(* Logix 5000 project; controller Drives_Line1 1756-L72 rev 20.13; software revision 20.04; part 17 of 21 *)
(* tags used below, declared in another part *)
   Bridle_04 : UDT_Bridle_3M;
   Bridle_04_FB_Diff : DINT;
   Bridle_04_FB_Update_Valid : BOOL;
   Bridle_04_Rev_mm : REAL;
   Bridle_04b_FBCounts_mm : REAL;
   Exit_Accu : UDT_Exit_Accu;
   ExitCtrl : UDT_Control_Zone;
   In_Config : UDT_Config;
   LineCmd : UDT_Commands_Line;
   Out_Feedbacks : UDT_Fdbks;
   Out_Status : UDT_Status;
   TaskInterval_ms : DINT;
   TestConfig_Exit_Accu : UDT_Config_Accu;
   TM3 : UDT_TM;
   zBridle_04b_Max_rev : REAL;
   zConfigFromMaster : BOOL;
   zPi : REAL;
(* P18_Exit_Accu, continued *)

ROUTINE R98_ToDrive   (* ladder *)
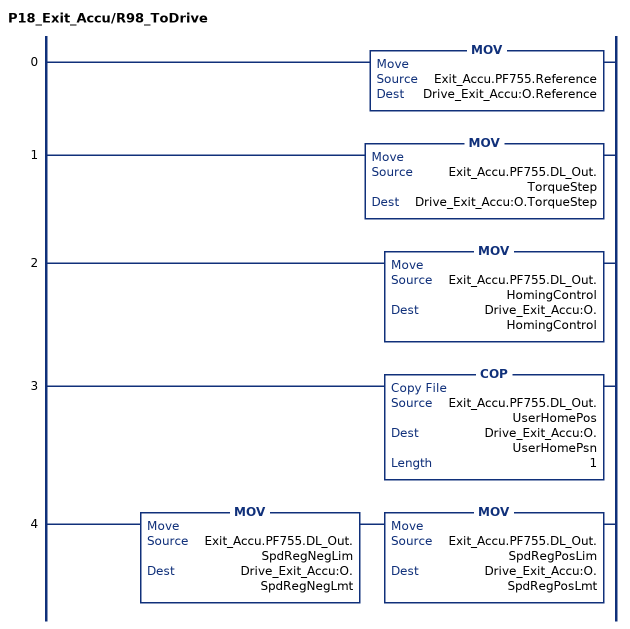
   0: MOV(Exit_Accu.PF755.Reference,Drive_Exit_Accu:O.Reference);
   1: MOV(Exit_Accu.PF755.DL_Out.TorqueStep,Drive_Exit_Accu:O.TorqueStep);
   2: MOV(Exit_Accu.PF755.DL_Out.HomingControl,Drive_Exit_Accu:O.HomingControl);
   3: COP(Exit_Accu.PF755.DL_Out.UserHomePos,Drive_Exit_Accu:O.UserHomePsn,1);
   4: MOV(Exit_Accu.PF755.DL_Out.SpdRegNegLim,Drive_Exit_Accu:O.SpdRegNegLmt)MOV(Exit_Accu.PF755.DL_Out.SpdRegPosLim,Drive_Exit_Accu:O.SpdRegPosLmt);
END_ROUTINE

ROUTINE R999_Test   (* ladder *)
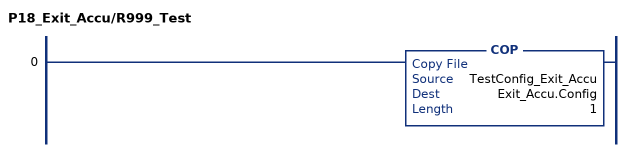
   0: COP(TestConfig_Exit_Accu,Exit_Accu.Config,1);
END_ROUTINE

ROUTINE R99_To_Master   (* ladder *)
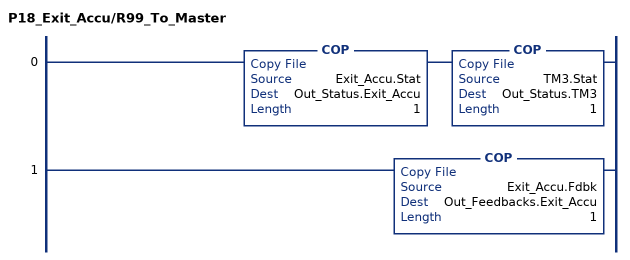
   0: COP(Exit_Accu.Stat,Out_Status.Exit_Accu,1)COP(TM3.Stat,Out_Status.TM3,1);
   1: COP(Exit_Accu.Fdbk,Out_Feedbacks.Exit_Accu,1);
END_ROUTINE
END_PROGRAM

PROGRAM P19_Bridle_04   (* main routine R00_Main *)
VAR
   ADD_01 : FBD_MATH := (SourceA := 0.0679603, Dest := 0.0679603);
   ADD_02 : FBD_MATH;
   BNOT_01 : FBD_BOOLEAN_NOT := (In := 1);
   BNOT_02 : FBD_BOOLEAN_NOT := (Out := 1);
   BOR_01 : FBD_BOOLEAN_OR := (In1 := 1, Out := 1);
   Bridle_04_FB_Count_Old : DINT := 7917204;
   Bridle_04_Max_FBcounts : REAL := 5120.0;
   Bridle_04_SpdTrimMPS : REAL;
   Bridle_04_SpdTrimPct : REAL;
   Bridle_04a_RPMPerMPS : REAL := 3303.7466;
   Bridle_04b_RPMPerMPS : REAL := 3085.579;
   Bridle_04c_RPMPerMPS : REAL := 2662.344;
   DIV_01 : FBD_MATH := (SourceB := 100.0);
   EQU_01 : FBD_COMPARE := (SourceA := 0.084748514);
   IO_State_Bridle_04a : INT := 4;
   IO_State_Bridle_04b : INT := 4;
   IO_State_Bridle_04c : INT := 4;
   IO_State_Tmp_Bridle_04a : INT := 16384;
   IO_State_Tmp_Bridle_04b : INT := 16384;
   IO_State_Tmp_Bridle_04c : INT := 16384;
   MUL_01 : FBD_MATH := (SourceB := 3085.579);
   MUL_02 : FBD_MATH := (SourceB := 3303.7466);
   MUL_05 : FBD_MATH;
   MUL_06 : FBD_MATH := (SourceB := 2662.344);
   Ons : DINT;
   PI_02 : PROP_INT := (In := -2.3841858e-07, Initialize := 1, Kp := 0.25, Wld := 0.05, HighLimit := 2.5, LowLimit := -2.5, ShapeKpPlus := 1.0, ShapeKpMinus := 1.0, ShapeWldPlus := 1.0, ShapeWldMinus := 1.0, RTSTime := 1, DeltaT := 0.05);
   PulsReset_PID : TIMER := (PRE := 250);
   SCL_09 : SCALE := (InRawMax := 100.0, InRawMin := -100.0, InEUMax := 2.5, InEUMin := -2.5, Limiting := 1, Out := -2.3841858e-07);
   SUB_02 : FBD_MATH;
   TimeOn_PIDOn : TIMER := (PRE := 500);
   TofReset : TIMER := (PRE := 1000, ACC := 1000);
   TonNoResponse : TIMER[3] := ([0].PRE := 2500, [1].PRE := 2500, [2].PRE := 2500);
   zBridle_04_Ki_SpdTrim : REAL := 0.05;
   zBridle_04_Kp_SpdTrim : REAL := 0.25;
   zBridle_04_MaxTrimSpdTrim : REAL := 2.5;
   zBridle_04_MinTrimSpdTrim : REAL := -2.5;
   zBridle_04b_EncRes : REAL := 4096.0;
END_VAR

ROUTINE R00_Main   (* ladder *)
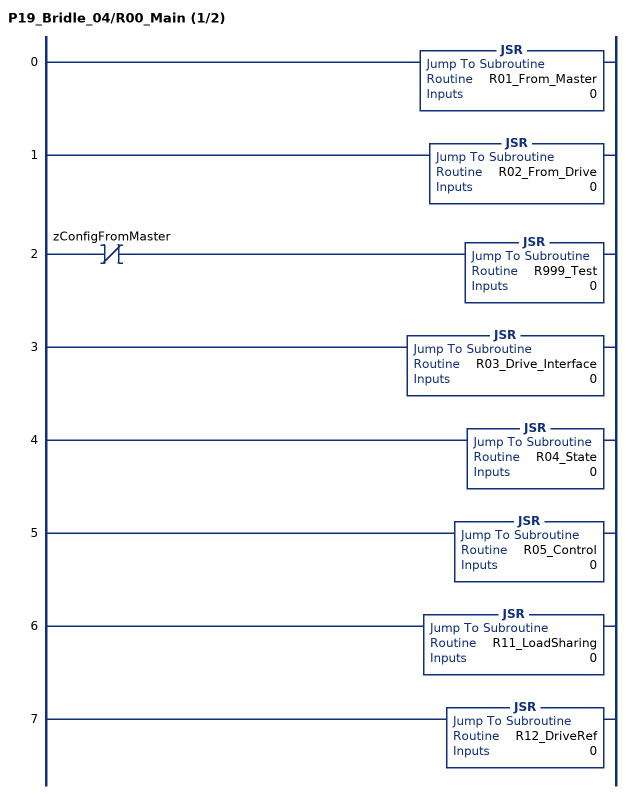
   0: JSR(R01_From_Master,0);
   1: JSR(R02_From_Drive,0);
   2: XIO(zConfigFromMaster)JSR(R999_Test,0);
   3: JSR(R03_Drive_Interface,0);
   4: JSR(R04_State,0);
   5: JSR(R05_Control,0);
   6: JSR(R11_LoadSharing,0);
   7: JSR(R12_DriveRef,0);
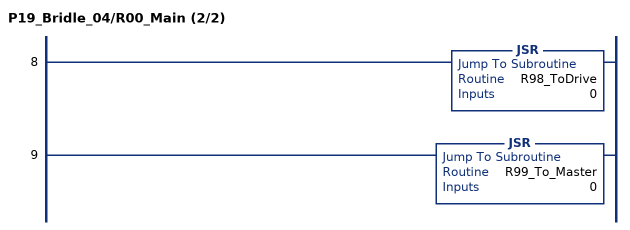
   8: JSR(R98_ToDrive,0);
   9: JSR(R99_To_Master,0);
END_ROUTINE

ROUTINE R01_From_Master   (* ladder *)
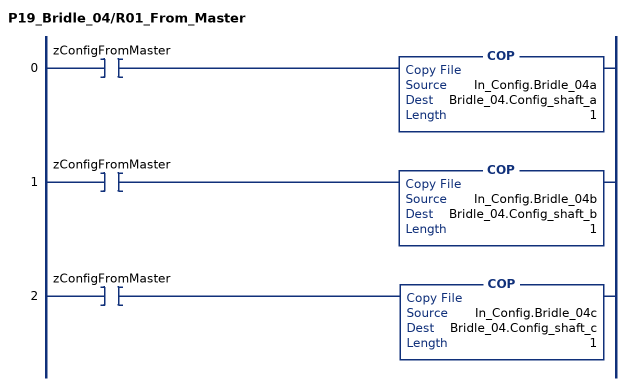
   0: XIC(zConfigFromMaster)COP(In_Config.Bridle_04a,Bridle_04.Config_shaft_a,1);
   1: XIC(zConfigFromMaster)COP(In_Config.Bridle_04b,Bridle_04.Config_shaft_b,1);
   2: XIC(zConfigFromMaster)COP(In_Config.Bridle_04c,Bridle_04.Config_shaft_c,1);
END_ROUTINE

ROUTINE R02_From_Drive   (* ladder *)
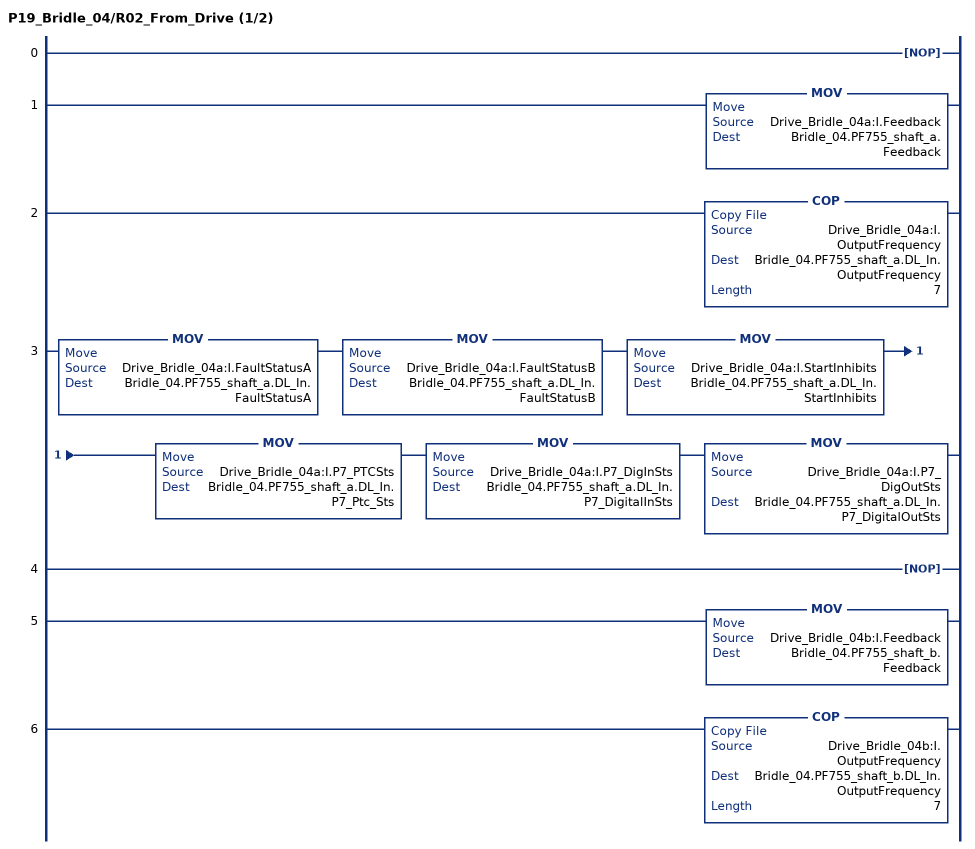
   0: NOP();
   1: MOV(Drive_Bridle_04a:I.Feedback,Bridle_04.PF755_shaft_a.Feedback);
   2: COP(Drive_Bridle_04a:I.OutputFrequency,Bridle_04.PF755_shaft_a.DL_In.OutputFrequency,7);
   3: MOV(Drive_Bridle_04a:I.FaultStatusA,Bridle_04.PF755_shaft_a.DL_In.FaultStatusA)MOV(Drive_Bridle_04a:I.FaultStatusB,Bridle_04.PF755_shaft_a.DL_In.FaultStatusB)MOV(Drive_Bridle_04a:I.StartInhibits,Bridle_04.PF755_shaft_a.DL_In.StartInhibits)MOV(Drive_Bridle_04a:I.P7_PTCSts,Bridle_04.PF755_shaft_a.DL_In.P7_Ptc_Sts)MOV(Drive_Bridle_04a:I.P7_DigInSts,Bridle_04.PF755_shaft_a.DL_In.P7_DigitalInSts)MOV(Drive_Bridle_04a:I.P7_DigOutSts,Bridle_04.PF755_shaft_a.DL_In.P7_DigitalOutSts);
   4: NOP();
   5: MOV(Drive_Bridle_04b:I.Feedback,Bridle_04.PF755_shaft_b.Feedback);
   6: COP(Drive_Bridle_04b:I.OutputFrequency,Bridle_04.PF755_shaft_b.DL_In.OutputFrequency,7);
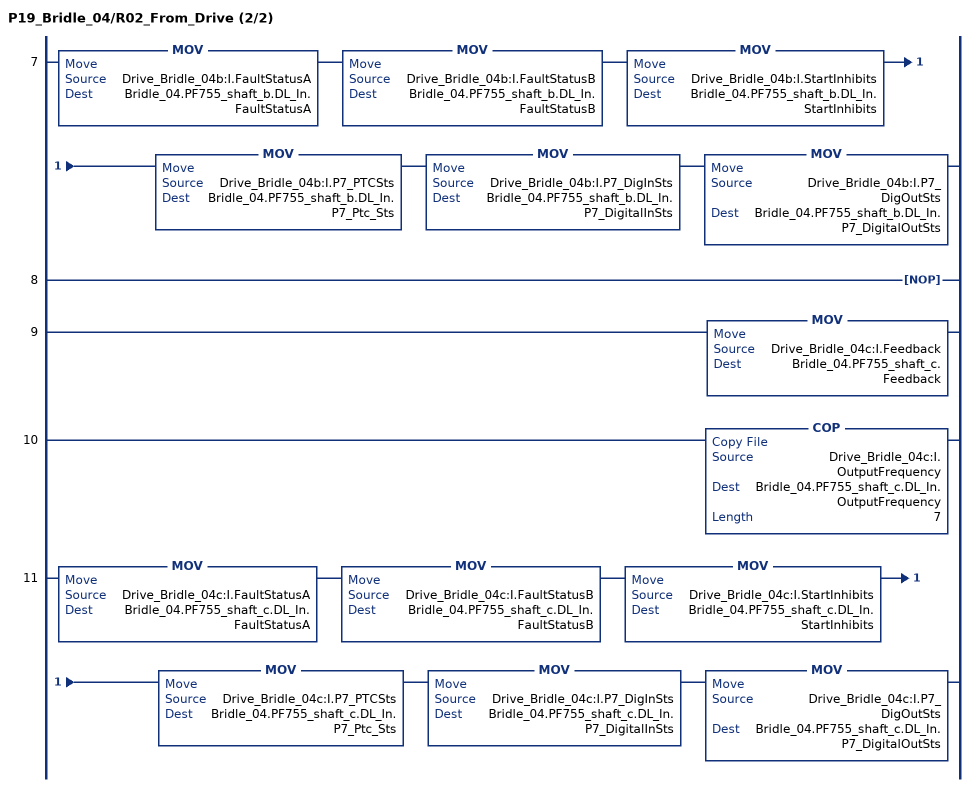
   7: MOV(Drive_Bridle_04b:I.FaultStatusA,Bridle_04.PF755_shaft_b.DL_In.FaultStatusA)MOV(Drive_Bridle_04b:I.FaultStatusB,Bridle_04.PF755_shaft_b.DL_In.FaultStatusB)MOV(Drive_Bridle_04b:I.StartInhibits,Bridle_04.PF755_shaft_b.DL_In.StartInhibits)MOV(Drive_Bridle_04b:I.P7_PTCSts,Bridle_04.PF755_shaft_b.DL_In.P7_Ptc_Sts)MOV(Drive_Bridle_04b:I.P7_DigInSts,Bridle_04.PF755_shaft_b.DL_In.P7_DigitalInSts)MOV(Drive_Bridle_04b:I.P7_DigOutSts,Bridle_04.PF755_shaft_b.DL_In.P7_DigitalOutSts);
   8: NOP();
   9: MOV(Drive_Bridle_04c:I.Feedback,Bridle_04.PF755_shaft_c.Feedback);
   10: COP(Drive_Bridle_04c:I.OutputFrequency,Bridle_04.PF755_shaft_c.DL_In.OutputFrequency,7);
   11: MOV(Drive_Bridle_04c:I.FaultStatusA,Bridle_04.PF755_shaft_c.DL_In.FaultStatusA)MOV(Drive_Bridle_04c:I.FaultStatusB,Bridle_04.PF755_shaft_c.DL_In.FaultStatusB)MOV(Drive_Bridle_04c:I.StartInhibits,Bridle_04.PF755_shaft_c.DL_In.StartInhibits)MOV(Drive_Bridle_04c:I.P7_PTCSts,Bridle_04.PF755_shaft_c.DL_In.P7_Ptc_Sts)MOV(Drive_Bridle_04c:I.P7_DigInSts,Bridle_04.PF755_shaft_c.DL_In.P7_DigitalInSts)MOV(Drive_Bridle_04c:I.P7_DigOutSts,Bridle_04.PF755_shaft_c.DL_In.P7_DigitalOutSts);
END_ROUTINE

ROUTINE R03_Drive_Interface   (* ladder *)
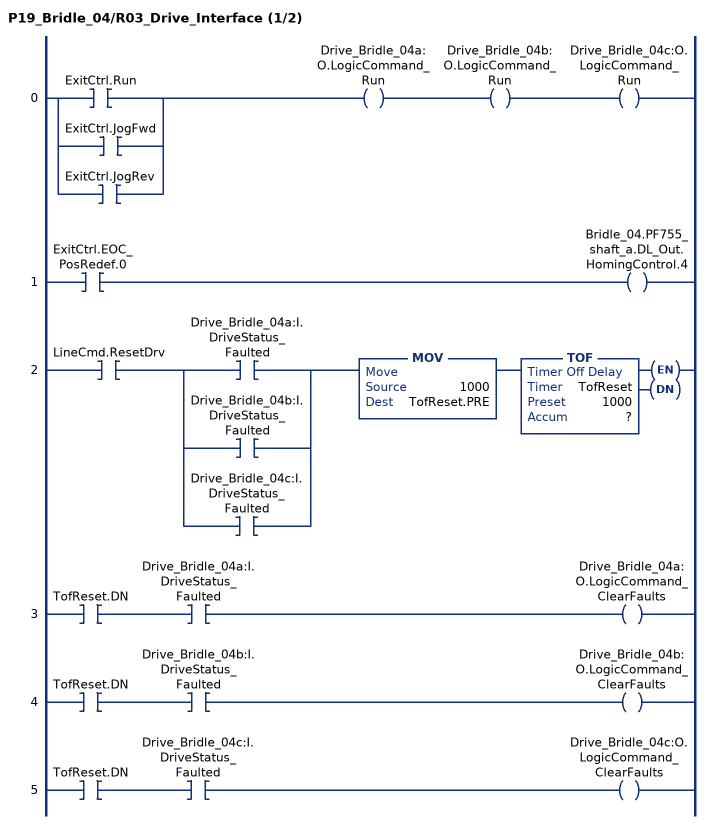
   0: [XIC(ExitCtrl.Run) ,XIC(ExitCtrl.JogFwd) ,XIC(ExitCtrl.JogRev) ]OTE(Drive_Bridle_04a:O.LogicCommand_Run)OTE(Drive_Bridle_04b:O.LogicCommand_Run)OTE(Drive_Bridle_04c:O.LogicCommand_Run);
   1: XIC(ExitCtrl.EOC_PosRedef.0)OTE(Bridle_04.PF755_shaft_a.DL_Out.HomingControl.4);
   2: XIC(LineCmd.ResetDrv)[XIC(Drive_Bridle_04a:I.DriveStatus_Faulted) ,XIC(Drive_Bridle_04b:I.DriveStatus_Faulted) ,XIC(Drive_Bridle_04c:I.DriveStatus_Faulted) ]MOV(1000,TofReset.PRE)TOF(TofReset,?,?);
   3: XIC(TofReset.DN)XIC(Drive_Bridle_04a:I.DriveStatus_Faulted)OTE(Drive_Bridle_04a:O.LogicCommand_ClearFaults);
   4: XIC(TofReset.DN)XIC(Drive_Bridle_04b:I.DriveStatus_Faulted)OTE(Drive_Bridle_04b:O.LogicCommand_ClearFaults);
   5: XIC(TofReset.DN)XIC(Drive_Bridle_04c:I.DriveStatus_Faulted)OTE(Drive_Bridle_04c:O.LogicCommand_ClearFaults);
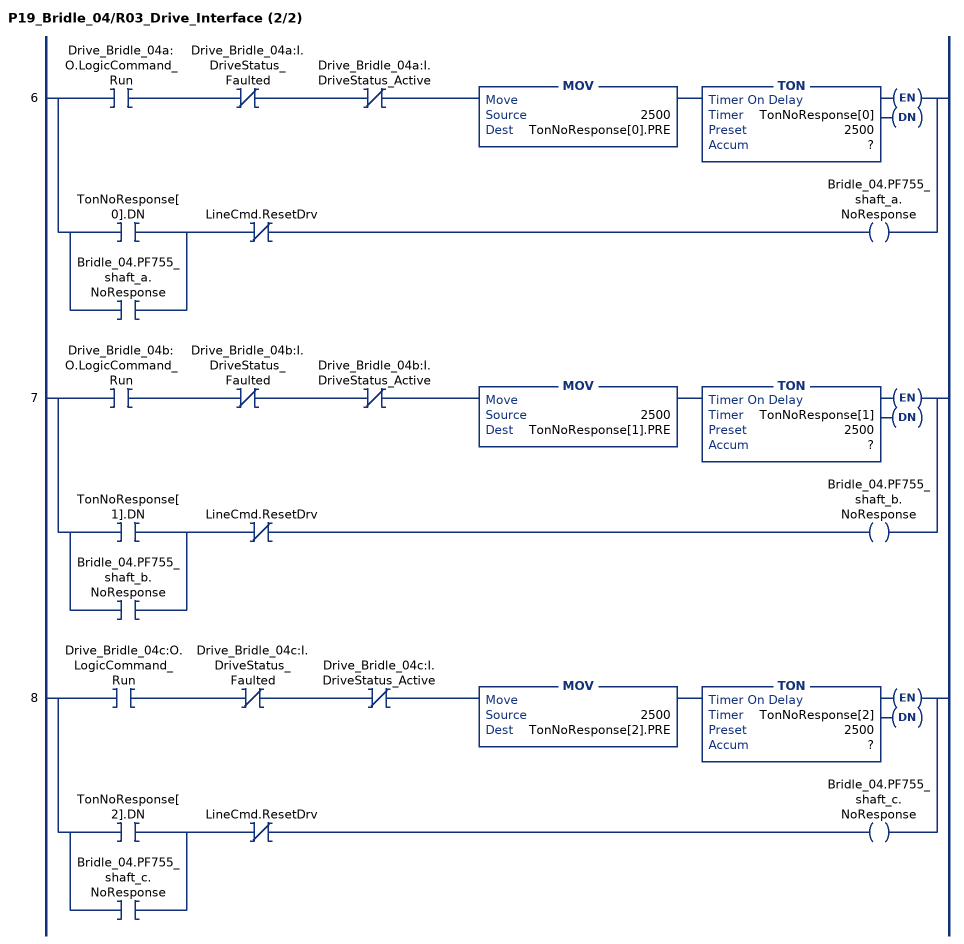
   6: [XIC(Drive_Bridle_04a:O.LogicCommand_Run) XIO(Drive_Bridle_04a:I.DriveStatus_Faulted) XIO(Drive_Bridle_04a:I.DriveStatus_Active) MOV(2500,TonNoResponse[0].PRE) TON(TonNoResponse[0],?,?) ,[XIC(TonNoResponse[0].DN) ,XIC(Bridle_04.PF755_shaft_a.NoResponse) ] XIO(LineCmd.ResetDrv) OTE(Bridle_04.PF755_shaft_a.NoResponse) ];
   7: [XIC(Drive_Bridle_04b:O.LogicCommand_Run) XIO(Drive_Bridle_04b:I.DriveStatus_Faulted) XIO(Drive_Bridle_04b:I.DriveStatus_Active) MOV(2500,TonNoResponse[1].PRE) TON(TonNoResponse[1],?,?) ,[XIC(TonNoResponse[1].DN) ,XIC(Bridle_04.PF755_shaft_b.NoResponse) ] XIO(LineCmd.ResetDrv) OTE(Bridle_04.PF755_shaft_b.NoResponse) ];
   8: [XIC(Drive_Bridle_04c:O.LogicCommand_Run) XIO(Drive_Bridle_04c:I.DriveStatus_Faulted) XIO(Drive_Bridle_04c:I.DriveStatus_Active) MOV(2500,TonNoResponse[2].PRE) TON(TonNoResponse[2],?,?) ,[XIC(TonNoResponse[2].DN) ,XIC(Bridle_04.PF755_shaft_c.NoResponse) ] XIO(LineCmd.ResetDrv) OTE(Bridle_04.PF755_shaft_c.NoResponse) ];
END_ROUTINE

ROUTINE R04_State   (* ladder *)
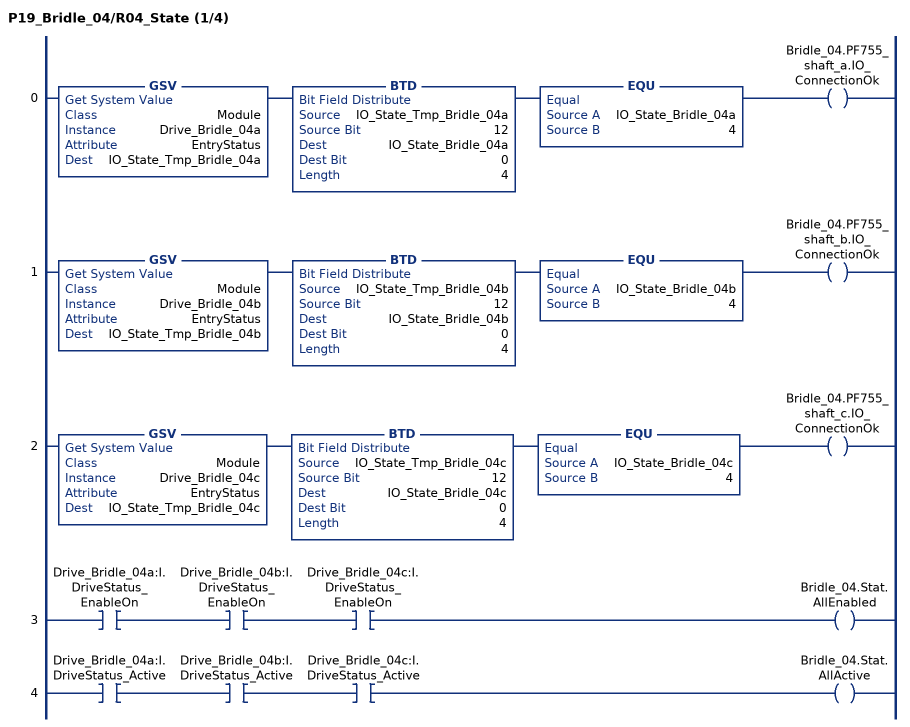
   0: GSV(Module,Drive_Bridle_04a,EntryStatus,IO_State_Tmp_Bridle_04a)BTD(IO_State_Tmp_Bridle_04a,12,IO_State_Bridle_04a,0,4)EQU(IO_State_Bridle_04a,4)OTE(Bridle_04.PF755_shaft_a.IO_ConnectionOk);
   1: GSV(Module,Drive_Bridle_04b,EntryStatus,IO_State_Tmp_Bridle_04b)BTD(IO_State_Tmp_Bridle_04b,12,IO_State_Bridle_04b,0,4)EQU(IO_State_Bridle_04b,4)OTE(Bridle_04.PF755_shaft_b.IO_ConnectionOk);
   2: GSV(Module,Drive_Bridle_04c,EntryStatus,IO_State_Tmp_Bridle_04c)BTD(IO_State_Tmp_Bridle_04c,12,IO_State_Bridle_04c,0,4)EQU(IO_State_Bridle_04c,4)OTE(Bridle_04.PF755_shaft_c.IO_ConnectionOk);
   3: XIC(Drive_Bridle_04a:I.DriveStatus_EnableOn)XIC(Drive_Bridle_04b:I.DriveStatus_EnableOn)XIC(Drive_Bridle_04c:I.DriveStatus_EnableOn)OTE(Bridle_04.Stat.AllEnabled);
   4: XIC(Drive_Bridle_04a:I.DriveStatus_Active)XIC(Drive_Bridle_04b:I.DriveStatus_Active)XIC(Drive_Bridle_04c:I.DriveStatus_Active)OTE(Bridle_04.Stat.AllActive);
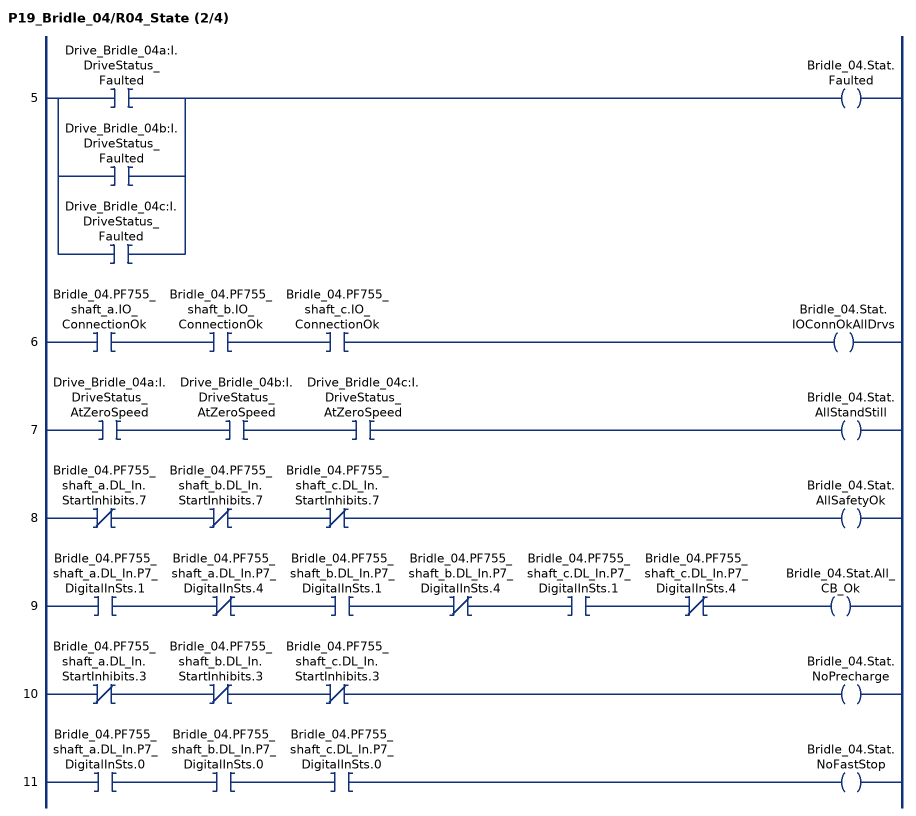
   5: [XIC(Drive_Bridle_04a:I.DriveStatus_Faulted) ,XIC(Drive_Bridle_04b:I.DriveStatus_Faulted) ,XIC(Drive_Bridle_04c:I.DriveStatus_Faulted) ]OTE(Bridle_04.Stat.Faulted);
   6: XIC(Bridle_04.PF755_shaft_a.IO_ConnectionOk)XIC(Bridle_04.PF755_shaft_b.IO_ConnectionOk)XIC(Bridle_04.PF755_shaft_c.IO_ConnectionOk)OTE(Bridle_04.Stat.IOConnOkAllDrvs);
   7: XIC(Drive_Bridle_04a:I.DriveStatus_AtZeroSpeed)XIC(Drive_Bridle_04b:I.DriveStatus_AtZeroSpeed)XIC(Drive_Bridle_04c:I.DriveStatus_AtZeroSpeed)OTE(Bridle_04.Stat.AllStandStill);
   8: XIO(Bridle_04.PF755_shaft_a.DL_In.StartInhibits.7)XIO(Bridle_04.PF755_shaft_b.DL_In.StartInhibits.7)XIO(Bridle_04.PF755_shaft_c.DL_In.StartInhibits.7)OTE(Bridle_04.Stat.AllSafetyOk);
   9: XIC(Bridle_04.PF755_shaft_a.DL_In.P7_DigitalInSts.1)XIO(Bridle_04.PF755_shaft_a.DL_In.P7_DigitalInSts.4)XIC(Bridle_04.PF755_shaft_b.DL_In.P7_DigitalInSts.1)XIO(Bridle_04.PF755_shaft_b.DL_In.P7_DigitalInSts.4)XIC(Bridle_04.PF755_shaft_c.DL_In.P7_DigitalInSts.1)XIO(Bridle_04.PF755_shaft_c.DL_In.P7_DigitalInSts.4)OTE(Bridle_04.Stat.All_CB_Ok);
   10: XIO(Bridle_04.PF755_shaft_a.DL_In.StartInhibits.3)XIO(Bridle_04.PF755_shaft_b.DL_In.StartInhibits.3)XIO(Bridle_04.PF755_shaft_c.DL_In.StartInhibits.3)OTE(Bridle_04.Stat.NoPrecharge);
   11: XIC(Bridle_04.PF755_shaft_a.DL_In.P7_DigitalInSts.0)XIC(Bridle_04.PF755_shaft_b.DL_In.P7_DigitalInSts.0)XIC(Bridle_04.PF755_shaft_c.DL_In.P7_DigitalInSts.0)OTE(Bridle_04.Stat.NoFastStop);
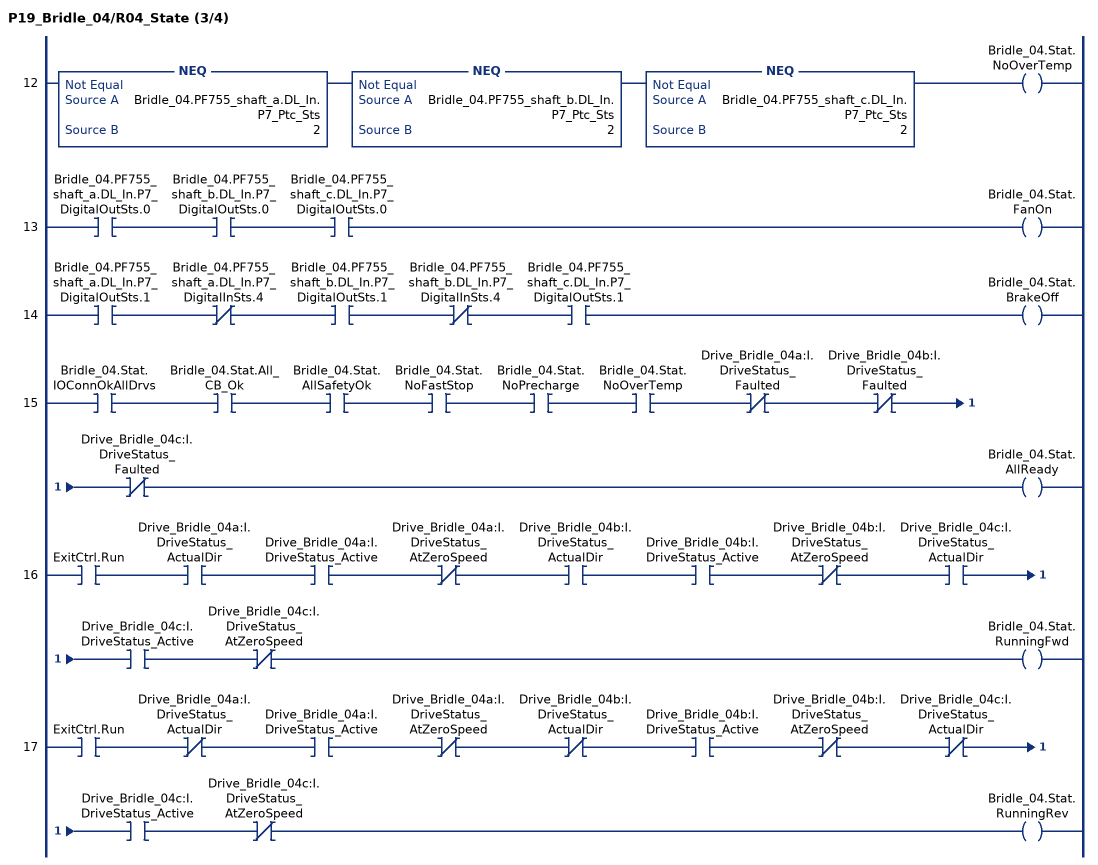
   12: NEQ(Bridle_04.PF755_shaft_a.DL_In.P7_Ptc_Sts,2)NEQ(Bridle_04.PF755_shaft_b.DL_In.P7_Ptc_Sts,2)NEQ(Bridle_04.PF755_shaft_c.DL_In.P7_Ptc_Sts,2)OTE(Bridle_04.Stat.NoOverTemp);
   13: XIC(Bridle_04.PF755_shaft_a.DL_In.P7_DigitalOutSts.0)XIC(Bridle_04.PF755_shaft_b.DL_In.P7_DigitalOutSts.0)XIC(Bridle_04.PF755_shaft_c.DL_In.P7_DigitalOutSts.0)OTE(Bridle_04.Stat.FanOn);
   14: XIC(Bridle_04.PF755_shaft_a.DL_In.P7_DigitalOutSts.1)XIO(Bridle_04.PF755_shaft_a.DL_In.P7_DigitalInSts.4)XIC(Bridle_04.PF755_shaft_b.DL_In.P7_DigitalOutSts.1)XIO(Bridle_04.PF755_shaft_b.DL_In.P7_DigitalInSts.4)XIC(Bridle_04.PF755_shaft_c.DL_In.P7_DigitalOutSts.1)OTE(Bridle_04.Stat.BrakeOff);
   15: XIC(Bridle_04.Stat.IOConnOkAllDrvs)XIC(Bridle_04.Stat.All_CB_Ok)XIC(Bridle_04.Stat.AllSafetyOk)XIC(Bridle_04.Stat.NoFastStop)XIC(Bridle_04.Stat.NoPrecharge)XIC(Bridle_04.Stat.NoOverTemp)XIO(Drive_Bridle_04a:I.DriveStatus_Faulted)XIO(Drive_Bridle_04b:I.DriveStatus_Faulted)XIO(Drive_Bridle_04c:I.DriveStatus_Faulted)OTE(Bridle_04.Stat.AllReady);
   16: XIC(ExitCtrl.Run)XIC(Drive_Bridle_04a:I.DriveStatus_ActualDir)XIC(Drive_Bridle_04a:I.DriveStatus_Active)XIO(Drive_Bridle_04a:I.DriveStatus_AtZeroSpeed)XIC(Drive_Bridle_04b:I.DriveStatus_ActualDir)XIC(Drive_Bridle_04b:I.DriveStatus_Active)XIO(Drive_Bridle_04b:I.DriveStatus_AtZeroSpeed)XIC(Drive_Bridle_04c:I.DriveStatus_ActualDir)XIC(Drive_Bridle_04c:I.DriveStatus_Active)XIO(Drive_Bridle_04c:I.DriveStatus_AtZeroSpeed)OTE(Bridle_04.Stat.RunningFwd);
   17: XIC(ExitCtrl.Run)XIO(Drive_Bridle_04a:I.DriveStatus_ActualDir)XIC(Drive_Bridle_04a:I.DriveStatus_Active)XIO(Drive_Bridle_04a:I.DriveStatus_AtZeroSpeed)XIO(Drive_Bridle_04b:I.DriveStatus_ActualDir)XIC(Drive_Bridle_04b:I.DriveStatus_Active)XIO(Drive_Bridle_04b:I.DriveStatus_AtZeroSpeed)XIO(Drive_Bridle_04c:I.DriveStatus_ActualDir)XIC(Drive_Bridle_04c:I.DriveStatus_Active)XIO(Drive_Bridle_04c:I.DriveStatus_AtZeroSpeed)OTE(Bridle_04.Stat.RunningRev);
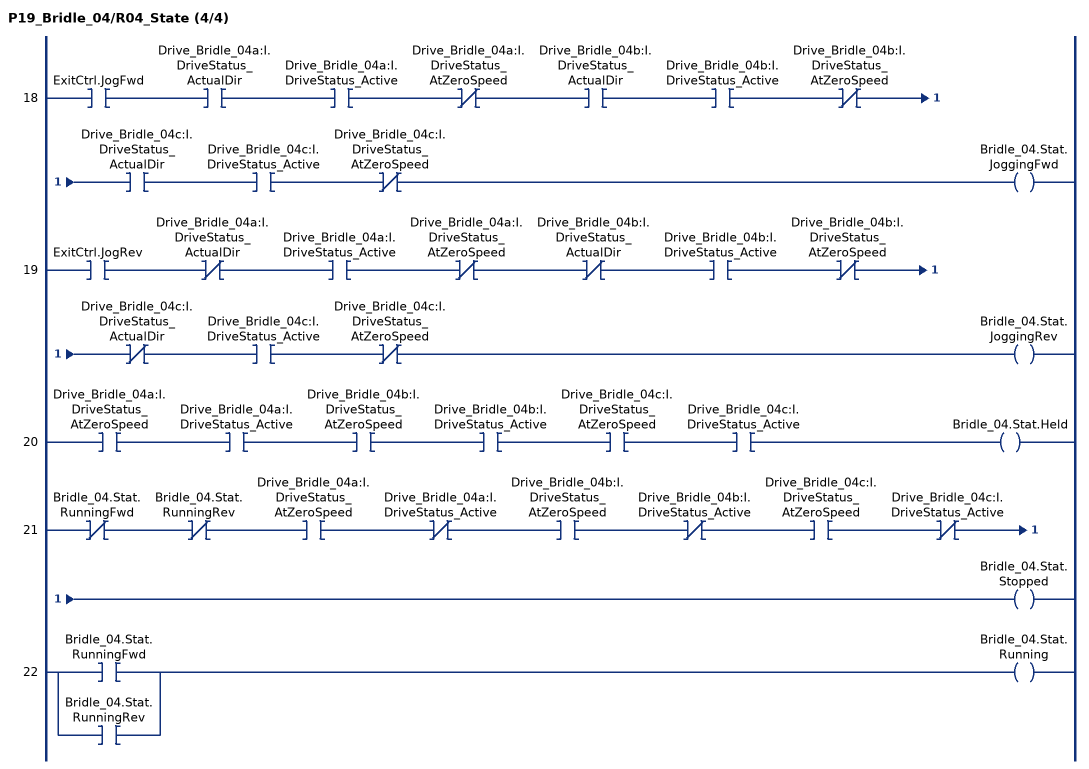
   18: XIC(ExitCtrl.JogFwd)XIC(Drive_Bridle_04a:I.DriveStatus_ActualDir)XIC(Drive_Bridle_04a:I.DriveStatus_Active)XIO(Drive_Bridle_04a:I.DriveStatus_AtZeroSpeed)XIC(Drive_Bridle_04b:I.DriveStatus_ActualDir)XIC(Drive_Bridle_04b:I.DriveStatus_Active)XIO(Drive_Bridle_04b:I.DriveStatus_AtZeroSpeed)XIC(Drive_Bridle_04c:I.DriveStatus_ActualDir)XIC(Drive_Bridle_04c:I.DriveStatus_Active)XIO(Drive_Bridle_04c:I.DriveStatus_AtZeroSpeed)OTE(Bridle_04.Stat.JoggingFwd);
   19: XIC(ExitCtrl.JogRev)XIO(Drive_Bridle_04a:I.DriveStatus_ActualDir)XIC(Drive_Bridle_04a:I.DriveStatus_Active)XIO(Drive_Bridle_04a:I.DriveStatus_AtZeroSpeed)XIO(Drive_Bridle_04b:I.DriveStatus_ActualDir)XIC(Drive_Bridle_04b:I.DriveStatus_Active)XIO(Drive_Bridle_04b:I.DriveStatus_AtZeroSpeed)XIO(Drive_Bridle_04c:I.DriveStatus_ActualDir)XIC(Drive_Bridle_04c:I.DriveStatus_Active)XIO(Drive_Bridle_04c:I.DriveStatus_AtZeroSpeed)OTE(Bridle_04.Stat.JoggingRev);
   20: XIC(Drive_Bridle_04a:I.DriveStatus_AtZeroSpeed)XIC(Drive_Bridle_04a:I.DriveStatus_Active)XIC(Drive_Bridle_04b:I.DriveStatus_AtZeroSpeed)XIC(Drive_Bridle_04b:I.DriveStatus_Active)XIC(Drive_Bridle_04c:I.DriveStatus_AtZeroSpeed)XIC(Drive_Bridle_04c:I.DriveStatus_Active)OTE(Bridle_04.Stat.Held);
   21: XIO(Bridle_04.Stat.RunningFwd)XIO(Bridle_04.Stat.RunningRev)XIC(Drive_Bridle_04a:I.DriveStatus_AtZeroSpeed)XIO(Drive_Bridle_04a:I.DriveStatus_Active)XIC(Drive_Bridle_04b:I.DriveStatus_AtZeroSpeed)XIO(Drive_Bridle_04b:I.DriveStatus_Active)XIC(Drive_Bridle_04c:I.DriveStatus_AtZeroSpeed)XIO(Drive_Bridle_04c:I.DriveStatus_Active)OTE(Bridle_04.Stat.Stopped);
   22: [XIC(Bridle_04.Stat.RunningFwd) ,XIC(Bridle_04.Stat.RunningRev) ]OTE(Bridle_04.Stat.Running);
END_ROUTINE

ROUTINE R05_Control   (* ladder *)
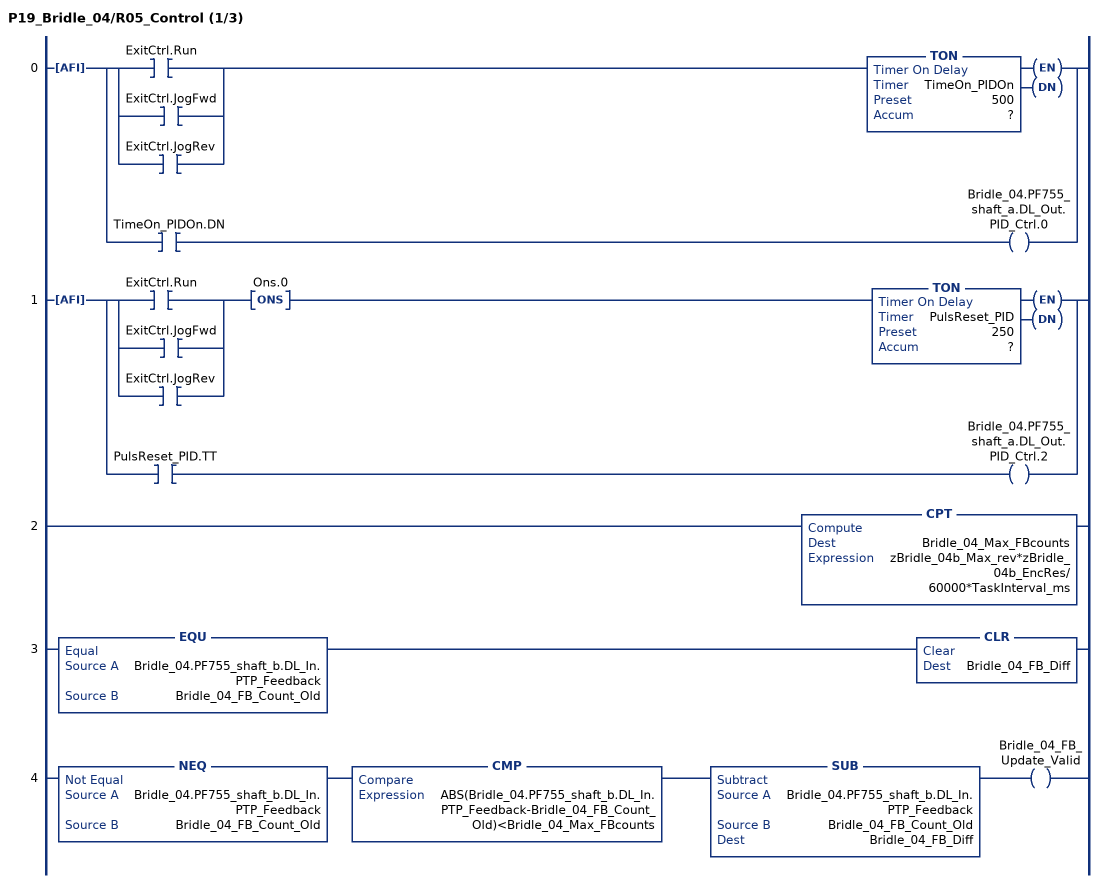
   0: AFI()[[XIC(ExitCtrl.Run) ,XIC(ExitCtrl.JogFwd) ,XIC(ExitCtrl.JogRev) ] TON(TimeOn_PIDOn,?,?) ,XIC(TimeOn_PIDOn.DN) OTE(Bridle_04.PF755_shaft_a.DL_Out.PID_Ctrl.0) ];
   1: AFI()[[XIC(ExitCtrl.Run) ,XIC(ExitCtrl.JogFwd) ,XIC(ExitCtrl.JogRev) ] ONS(Ons.0) TON(PulsReset_PID,?,?) ,XIC(PulsReset_PID.TT) OTE(Bridle_04.PF755_shaft_a.DL_Out.PID_Ctrl.2) ];
   2: CPT(Bridle_04_Max_FBcounts,zBridle_04b_Max_rev*zBridle_04b_EncRes/60000*TaskInterval_ms);
   3: EQU(Bridle_04.PF755_shaft_b.DL_In.PTP_Feedback,Bridle_04_FB_Count_Old)CLR(Bridle_04_FB_Diff);
   4: NEQ(Bridle_04.PF755_shaft_b.DL_In.PTP_Feedback,Bridle_04_FB_Count_Old)CMP(ABS(Bridle_04.PF755_shaft_b.DL_In.PTP_Feedback-Bridle_04_FB_Count_Old)<Bridle_04_Max_FBcounts)SUB(Bridle_04.PF755_shaft_b.DL_In.PTP_Feedback,Bridle_04_FB_Count_Old,Bridle_04_FB_Diff)OTE(Bridle_04_FB_Update_Valid);
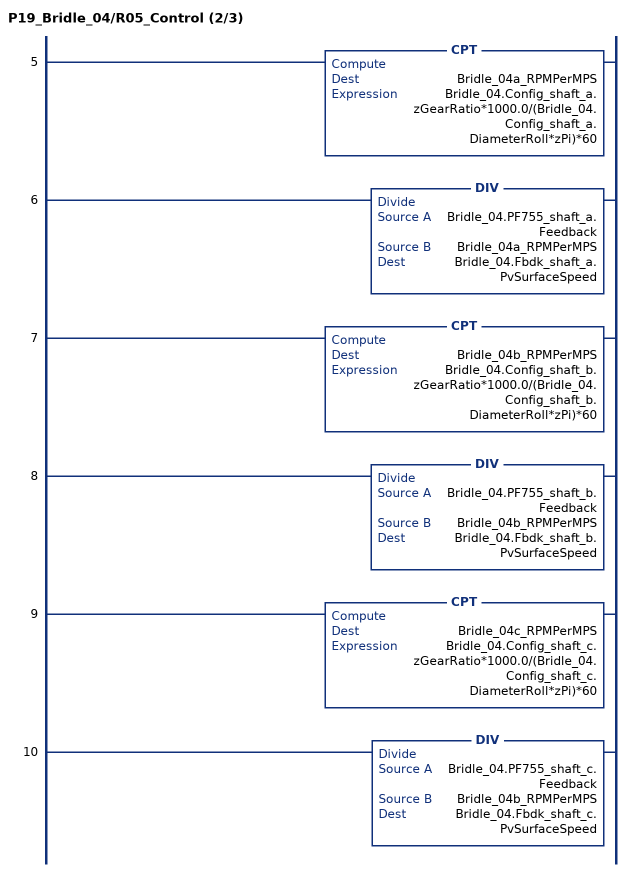
   5: CPT(Bridle_04a_RPMPerMPS,Bridle_04.Config_shaft_a.zGearRatio*1000.0/(Bridle_04.Config_shaft_a.DiameterRoll*zPi)*60);
   6: DIV(Bridle_04.PF755_shaft_a.Feedback,Bridle_04a_RPMPerMPS,Bridle_04.Fbdk_shaft_a.PvSurfaceSpeed);
   7: CPT(Bridle_04b_RPMPerMPS,Bridle_04.Config_shaft_b.zGearRatio*1000.0/(Bridle_04.Config_shaft_b.DiameterRoll*zPi)*60);
   8: DIV(Bridle_04.PF755_shaft_b.Feedback,Bridle_04b_RPMPerMPS,Bridle_04.Fbdk_shaft_b.PvSurfaceSpeed);
   9: CPT(Bridle_04c_RPMPerMPS,Bridle_04.Config_shaft_c.zGearRatio*1000.0/(Bridle_04.Config_shaft_c.DiameterRoll*zPi)*60);
   10: DIV(Bridle_04.PF755_shaft_c.Feedback,Bridle_04b_RPMPerMPS,Bridle_04.Fbdk_shaft_c.PvSurfaceSpeed);
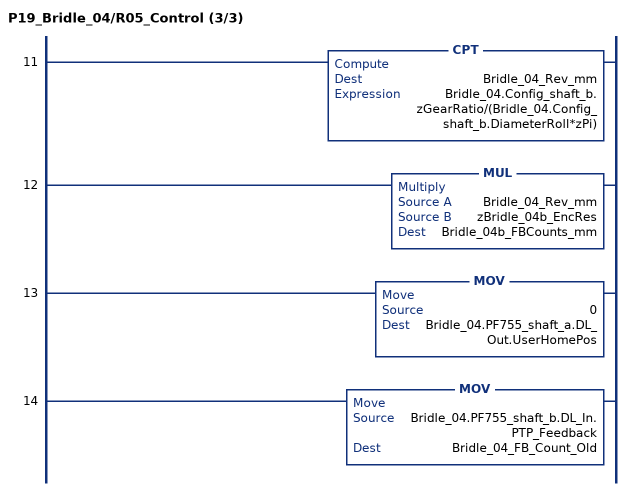
   11: CPT(Bridle_04_Rev_mm,Bridle_04.Config_shaft_b.zGearRatio/(Bridle_04.Config_shaft_b.DiameterRoll*zPi));
   12: MUL(Bridle_04_Rev_mm,zBridle_04b_EncRes,Bridle_04b_FBCounts_mm);
   13: MOV(0,Bridle_04.PF755_shaft_a.DL_Out.UserHomePos);
   14: MOV(Bridle_04.PF755_shaft_b.DL_In.PTP_Feedback,Bridle_04_FB_Count_Old);
END_ROUTINE

ROUTINE R11_LoadSharing   (* function block diagram *)
   SHEET 1   // Load sharing speed trim percentage
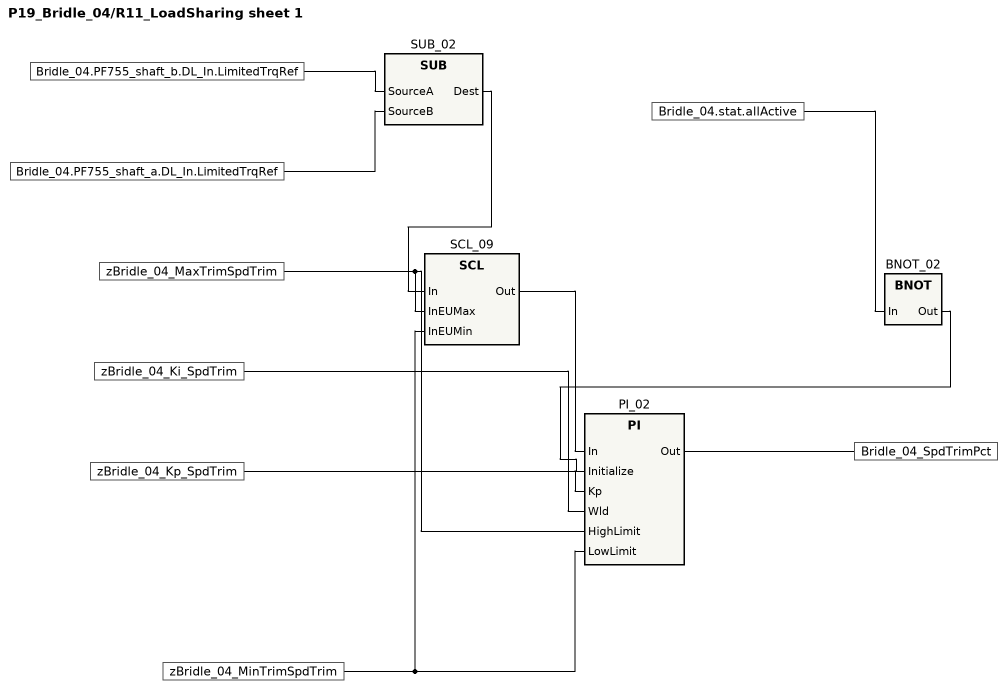
   SUB_02 : SUB(SourceA := Bridle_04.PF755_shaft_b.DL_In.LimitedTrqRef, SourceB := Bridle_04.PF755_shaft_a.DL_In.LimitedTrqRef);
   SCL_09 : SCL(In := SUB_02.Dest, InEUMax := zBridle_04_MaxTrimSpdTrim, InEUMin := zBridle_04_MinTrimSpdTrim);
   BNOT_02 : BNOT(In := Bridle_04.stat.allActive);
   PI_02 : PI(In := SCL_09.Out, Initialize := BNOT_02.Out, Kp := zBridle_04_Kp_SpdTrim, Wld := zBridle_04_Ki_SpdTrim, HighLimit := zBridle_04_MaxTrimSpdTrim, LowLimit := zBridle_04_MinTrimSpdTrim);
   Bridle_04_SpdTrimPct := PI_02.Out;
   SHEET 2   // Calculate speed trim mps
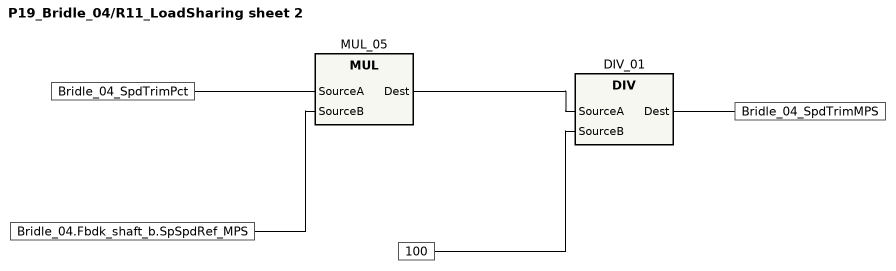
   MUL_05 : MUL(SourceA := Bridle_04_SpdTrimPct, SourceB := Bridle_04.Fbdk_shaft_b.SpSpdRef_MPS);
   DIV_01 : DIV(SourceA := MUL_05.Dest, SourceB := 100);
   Bridle_04_SpdTrimMPS := DIV_01.Dest;
END_ROUTINE
